FUNCTION_BLOCK FB_Auswertung
VAR_INPUT
	I_RNr				:INT;
	I_ConnectionHdl		:DWORD;
	I_NameSpace			:STRING(MAX_STRING_LENGTH);
	I_CW				:RezeptControlWord;
	I_SW				:RezeptStatusWord;
	I_SysSW				:SystemStatusWord;
	I_SekCW				:SekControlWord;
END_VAR

VAR_OUTPUT
	O_Verbunden			:BOOL;
	O_SysSW				:SystemStatusWord;
	O_SekCW				:SekControlWord;
	O_Error				:BOOL;
	O_ErrorID			:DWORD;
END_VAR

VAR
	OPC_Status			:INT;
	SysSW					:SystemStatusWord;			// Variable für Handling von SystemStatusWord
	SekCW					:SekControlWord;			// Variable für Handling von Start von sekundär Reaktor
	
	// Instanziierung der Kommunikationsfunktionsblöcke
	NameSpaceInd		:UA_GetNamespaceIndex;
	Node				:UA_NodeGetHandle;
	NodeRelease			:UA_NodeReleaseHandle;
	Write				:UA_Write;
	
	// Instanziierung der relevanten Input-Variablen
	NodeID_SysSW			:ST_UANodeID;
	NodeID_SekCW			:ST_UANodeID;
	NodeIdentifier_SysSW	:STRING(MAX_STRING_LENGTH) := 'GVL_OPC_UA.SysSW';
	NodeIdentifier_SekCW	:STRING(MAX_STRING_LENGTH) := 'GVL_OPC_UA.SekCW';
	
	// Instanziierung der relevanten Output-Variablen
	NameSpaceIndex			:UINT;
	NodeHdl_SysSW			:DWORD;	
	NodeHdl_SekCW			:DWORD;
	
END_VAR

CASE OPC_Status OF 
	0:	// Idle
	
	//==================================================================================================
	1: // GetNameSpace - SystemStatusWord
		NameSpaceInd(Execute := TRUE,
				ConnectionHdl := I_ConnectionHdl,
				NameSpaceUri := I_NameSpace,
				Timeout := T#5S,
				NameSpaceIndex => NameSpaceIndex, 
				Error => O_Error, 
				ErrorID => O_ErrorID);
					
		IF NOT NameSpaceInd.Busy THEN
			NameSpaceInd(Execute := FALSE);
		END_IF
					
		IF NameSpaceInd.Error THEN
			O_Verbunden := FALSE;
			OPC_Status := 0;
		END_IF
		
		IF NameSpaceInd.Done THEN
			OPC_Status := 2;
		END_IF
	
	//==================================================================================================
	2: // GetNode - SystemStatusWord
		NodeID_SysSW.eIdentifierType := eUAIdentifierType_String;
		NodeID_SysSW.nNamespaceIndex := NameSpaceIndex;
		NodeID_SysSW.sIdentifier := NodeIdentifier_SysSW;
	
		Node(Execute := TRUE,
				ConnectionHdl := I_ConnectionHdl,
				NodeID := NodeID_SysSW,
				Timeout := T#5S,
				NodeHdl => NodeHdl_SysSW, 
				Error => O_Error, 
				ErrorID => O_ErrorID);

		IF NOT Node.Busy THEN
			Node(Execute := FALSE);
		END_IF 		
		
		IF Node.Error THEN
			OPC_Status := 0;
		END_IF
		
		IF Node.Done THEN
			OPC_Status := 3; 	
		END_IF
		
	//==================================================================================================
	3: // GetNode - SekControlWord
		NodeID_SekCW.eIdentifierType := eUAIdentifierType_String;
		NodeID_SekCW.nNamespaceIndex := NameSpaceIndex;
		NodeID_SekCW.sIdentifier := NodeIdentifier_SekCW;
	
		// Definieren von SW Node
		Node(Execute := TRUE,
				ConnectionHdl := I_ConnectionHdl,
				NodeID := NodeID_SekCW,
				Timeout := T#5S,
				NodeHdl => NodeHdl_SekCW, 
				Error => O_Error, 
				ErrorID => O_ErrorID);

		IF NOT Node.Busy THEN
			Node(Execute := FALSE);
		END_IF 		
	
	IF Node.Error THEN
		OPC_Status := 0;
	END_IF
	
	IF Node.Done THEN
		OPC_Status := 0;
		O_Verbunden := TRUE;	
	END_IF
	
	//==================================================================================================
	4: // Beschreiben von SystemStatusWord auf allen Reaktoren
	   // Definieren des Zustandes des SystemSatusWords
	   SysSW := I_SysSW;
	   
		CASE I_RNr OF 
			1:	SysSW.R1_Ready := I_SW.ReactReady;
				SysSW.R1_Activ := I_SW.ReactActiv;
				
			2:	SysSW.R2_Ready := I_SW.ReactReady;
				SysSW.R2_Activ := I_SW.ReactActiv;
				
			3:	SysSW.R3_Ready := I_SW.ReactReady;
				SysSW.R3_Activ := I_SW.ReactActiv;
				
			4:	SysSW.R4_Ready := I_SW.ReactReady;
				SysSW.R4_Activ := I_SW.ReactActiv;
				
			5:	SysSW.R5_Ready := I_SW.ReactReady;
				SysSW.R5_Activ := I_SW.ReactActiv;
				
			6:	SysSW.R6_Ready := I_SW.ReactReady;
				SysSW.R6_Activ := I_SW.ReactActiv;
				
			7:	SysSW.R7_Ready := I_SW.ReactReady;
				SysSW.R7_Activ := I_SW.ReactActiv;
		END_CASE
	
		// SystemStatusWord schreiben
		Write(Execute := TRUE,
			ConnectionHdl := I_ConnectionHdl,
			NodeHdl := NodeHdl_SysSW,
			pVariable := ADR(SysSW),
			cbData  := SIZEOF(SysSW),
			Timeout := T#5S,
			Error => O_Error,
			ErrorID => O_ErrorID);
			
		IF NOT Write.Busy THEN
			Write(Execute := FALSE);
		END_IF	
			
		IF Write.Error THEN
			OPC_Status := 0;
		END_IF
		
		IF Write.Done THEN
			OPC_Status := 0;
			O_SysSW := SysSW;
		END_IF	
	
	//==================================================================================================
	5: // Schreiben von Startvariablen für Sekundärreaktor
		SekCW := I_SekCW;
	
		CASE I_CW.Leitung OF
			0: SekCW.R1 := FALSE;
			   SekCW.R2 := FALSE;
			   SekCW.R3 := FALSE;
			   SekCW.R4 := FALSE;
			   SekCW.R5 := FALSE;
			   SekCW.R6 := FALSE;
			   SekCW.R7 := FALSE;
			   
			1: SekCW.R1 := TRUE;
			2: SekCW.R2 := TRUE;	
			3: SekCW.R3 := TRUE;
			4: SekCW.R4 := TRUE;
			5: SekCW.R5 := TRUE;
			6: SekCW.R6 := TRUE;
			7: SekCW.R7 := TRUE;
		END_CASE
	
		// SystemStatusWord schreiben
		Write(Execute := TRUE,
			ConnectionHdl := I_ConnectionHdl,
			NodeHdl := NodeHdl_SekCW,
			pVariable := ADR(SekCW),
			cbData  := SIZEOF(SekCW),
			Timeout := T#5S,
			Error => O_Error,
			ErrorID => O_ErrorID);
		
		IF NOT Write.Busy THEN
			Write(Execute := FALSE);
		END_IF	
			
		IF Write.Error THEN
			OPC_Status := 0;
		END_IF
	
		IF Write.Done THEN
			OPC_Status := 0;
			O_SekCW := SekCW;
		END_IF	
		
	//==================================================================================================
	6: // ReleaseNode - SystemStatusWord
		NodeRelease(Execute := TRUE,
				ConnectionHdl := I_ConnectionHdl,
				NodeHdl := NodeHdl_SysSW,
				Timeout := T#5S,
				Error => O_Error,
				ErrorID => O_ErrorID);
	
		IF NOT NodeRelease.Busy THEN
			NodeRelease(Execute := FALSE);
		END_IF
		
		IF NodeRelease.Error THEN
			OPC_Status := 0;
		END_IF
	
		IF NodeRelease.Done THEN
			OPC_Status := 7;
		END_IF		
	//==================================================================================================
	7: // ReleaseNode - SekControlWord
		NodeRelease(Execute := TRUE,
				ConnectionHdl := I_ConnectionHdl,
				NodeHdl := NodeHdl_SekCW,
				Timeout := T#5S,
				Error => O_Error,
				ErrorID => O_ErrorID);
	
		IF NOT NodeRelease.Busy THEN
			NodeRelease(Execute := FALSE);
		END_IF
		
		IF NodeRelease.Error THEN
			OPC_Status := 0;
		END_IF
	
		IF NodeRelease.Done THEN
			OPC_Status := 0;
		END_IF
END_CASE

METHOD M_STATUS_SEK : BOOL
VAR_INPUT
END_VAR
OPC_Status := 5;
END_METHOD

METHOD M_STATUS_SYSTEM : BOOL
VAR_INPUT
END_VAR
OPC_Status := 4;
END_METHOD

METHOD M_TRENNEN : BOOL
VAR_INPUT
END_VAR
OPC_Status := 6;
END_METHOD

METHOD M_VERBINDEN : BOOL
VAR_INPUT
END_VAR
OPC_Status := 1;
END_METHOD

END_FUNCTION_BLOCK

(* stored: Version 1.1.0.1, ProductVersion 3.1.4024.12
   POU FB_Auswertung: Id {0842150b-4601-4fae-871d-0c9147fd5aad}, SpecialFunc None
   Method M_STATUS_SEK: Id {bad8bb1c-0495-49d6-b646-cf414b9f672e}
   Method M_STATUS_SYSTEM: Id {9603de6b-8fe5-4482-ae8e-004d0e964aa2}
   Method M_TRENNEN: Id {bf136760-2fb3-4eb1-b732-6c62789e7908}
   Method M_VERBINDEN: Id {df7aed53-903a-4160-b680-3b353057e7b0} *)
